// Mitsubishi GX Works2 project: pr6   PLC: Q03UDV

PROGRAM MAIN
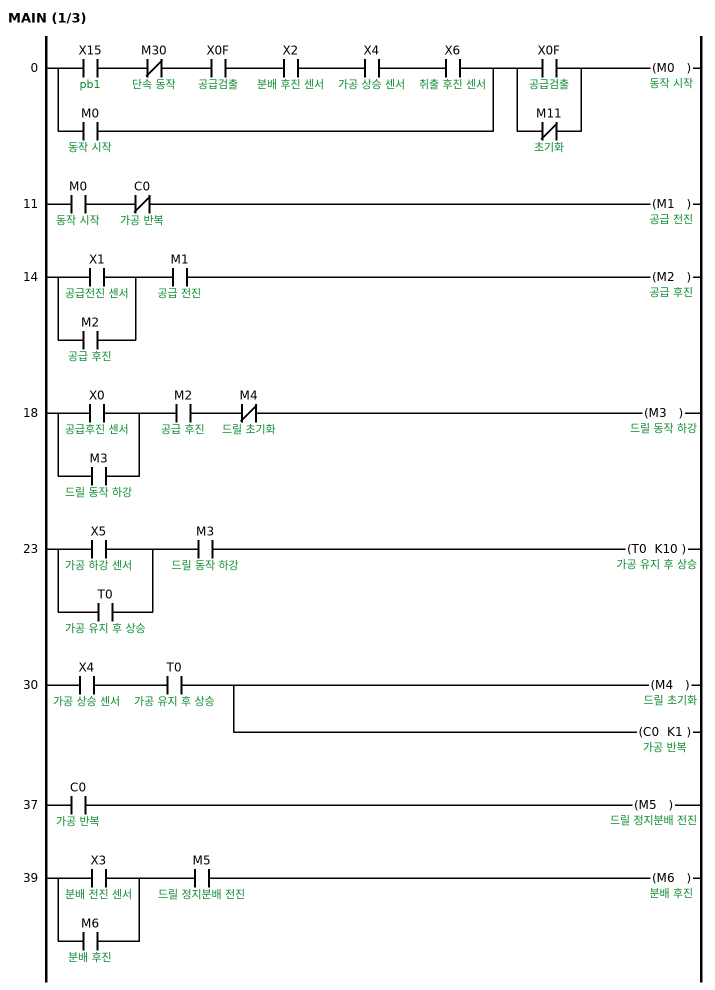
0     LD      X15  ; pb1
      ANI     M30  ; 단속 동작
      AND     X0F  ; 공급검출
      AND     X2  ; 분배 후진 센서
      AND     X4  ; 가공 상승 센서
      AND     X6  ; 취출 후진 센서
      OR      M0  ; 동작 시작
      LD      X0F  ; 공급검출
      ORI     M11  ; 초기화
      ANB
      OUT     M0  ; 동작 시작
11    LD      M0  ; 동작 시작
      ANI     C0  ; 가공 반복
      OUT     M1  ; 공급 전진
14    LD      X1  ; 공급전진 센서
      OR      M2  ; 공급 후진
      AND     M1  ; 공급 전진
      OUT     M2  ; 공급 후진
18    LD      X0  ; 공급후진 센서
      OR      M3  ; 드릴 동작 하강
      AND     M2  ; 공급 후진
      ANI     M4  ; 드릴 초기화
      OUT     M3  ; 드릴 동작 하강
23    LD      X5  ; 가공 하강 센서
      OR      T0  ; 가공 유지 후 상승
      AND     M3  ; 드릴 동작 하강
      OUT     T0 K10  ; 가공 유지 후 상승
30    LD      X4  ; 가공 상승 센서
      AND     T0  ; 가공 유지 후 상승
      OUT     M4  ; 드릴 초기화
      OUT     C0 K1  ; 가공 반복
37    LD      C0  ; 가공 반복
      OUT     M5  ; 드릴 정지분배 전진
39    LD      X3  ; 분배 전진 센서
      OR      M6  ; 분배 후진
      AND     M5  ; 드릴 정지분배 전진
      OUT     M6  ; 분배 후진
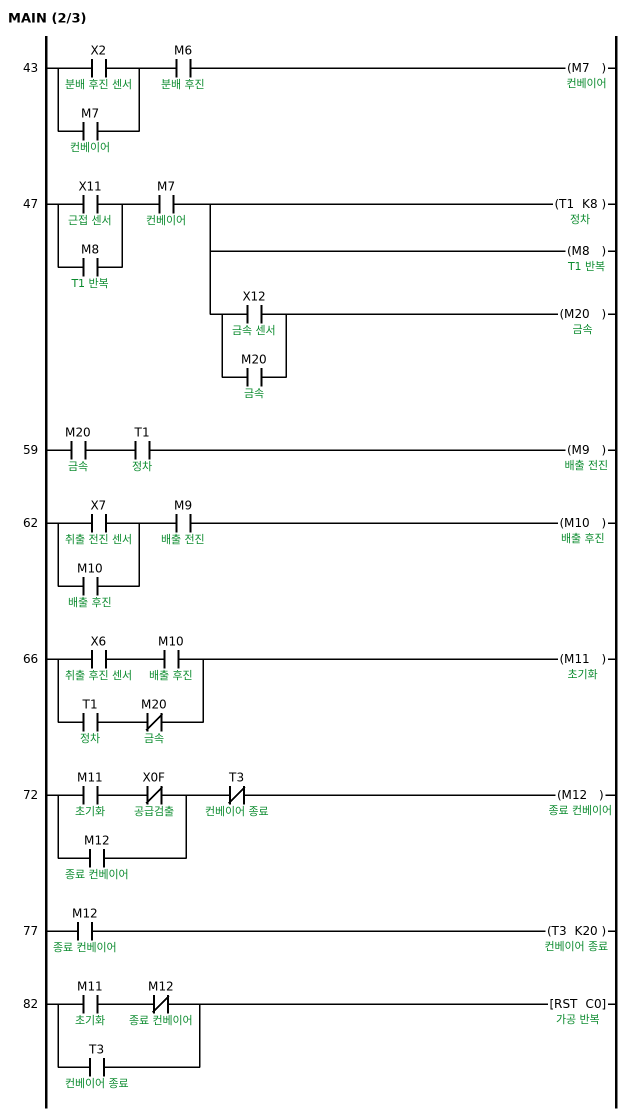
43    LD      X2  ; 분배 후진 센서
      OR      M7  ; 컨베이어
      AND     M6  ; 분배 후진
      OUT     M7  ; 컨베이어
47    LD      X11  ; 근접 센서
      OR      M8  ; T1 반복
      AND     M7  ; 컨베이어
      OUT     T1 K8  ; 정차
      OUT     M8  ; T1 반복
      LD      X12  ; 금속 센서
      OR      M20  ; 금속
      ANB
      OUT     M20  ; 금속
59    LD      M20  ; 금속
      AND     T1  ; 정차
      OUT     M9  ; 배출 전진
62    LD      X7  ; 취출 전진 센서
      OR      M10  ; 배출 후진
      AND     M9  ; 배출 전진
      OUT     M10  ; 배출 후진
66    LD      X6  ; 취출 후진 센서
      AND     M10  ; 배출 후진
      LD      T1  ; 정차
      ANI     M20  ; 금속
      ORB
      OUT     M11  ; 초기화
72    LD      M11  ; 초기화
      ANI     X0F  ; 공급검출
      OR      M12  ; 종료 컨베이어
      ANI     T3  ; 컨베이어 종료
      OUT     M12  ; 종료 컨베이어
77    LD      M12  ; 종료 컨베이어
      OUT     T3 K20  ; 컨베이어 종료
82    LD      M11  ; 초기화
      ANI     M12  ; 종료 컨베이어
      OR      T3  ; 컨베이어 종료
      RST     C0  ; 가공 반복
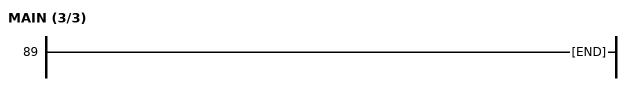
89    END
END_PROGRAM

PROGRAM OUTPUT
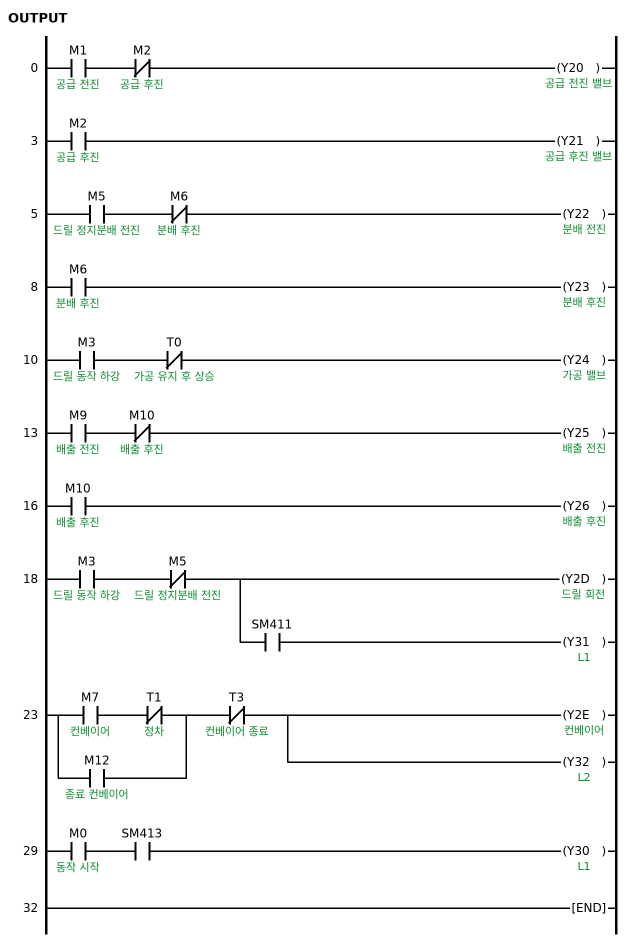
0     LD      M1  ; 공급 전진
      ANI     M2  ; 공급 후진
      OUT     Y20  ; 공급 전진 밸브
3     LD      M2  ; 공급 후진
      OUT     Y21  ; 공급 후진 밸브
5     LD      M5  ; 드릴 정지분배 전진
      ANI     M6  ; 분배 후진
      OUT     Y22  ; 분배 전진
8     LD      M6  ; 분배 후진
      OUT     Y23  ; 분배 후진
10    LD      M3  ; 드릴 동작 하강
      ANI     T0  ; 가공 유지 후 상승
      OUT     Y24  ; 가공 밸브
13    LD      M9  ; 배출 전진
      ANI     M10  ; 배출 후진
      OUT     Y25  ; 배출 전진
16    LD      M10  ; 배출 후진
      OUT     Y26  ; 배출 후진
18    LD      M3  ; 드릴 동작 하강
      ANI     M5  ; 드릴 정지분배 전진
      OUT     Y2D  ; 드릴 회전
      AND     SM411
      OUT     Y31  ; L1
23    LD      M7  ; 컨베이어
      ANI     T1  ; 정차
      OR      M12  ; 종료 컨베이어
      ANI     T3  ; 컨베이어 종료
      OUT     Y2E  ; 컨베이어
      OUT     Y32  ; L2
29    LD      M0  ; 동작 시작
      AND     SM413
      OUT     Y30  ; L1
32    END
END_PROGRAM

// device comments not shown above
X10  ; 근접 센서
X16  ; PB2
X18  ; pb4
M15  ; 초기화 묶음
M21  ; 프로그램 초기화
M40  ; 종료 버튼
M41  ; 종료조건
M100  ; 종료 버튼 눌림
M101  ; 전체 종료
T2  ; 드릴 유지
T4  ; 취출 복귀
T5  ; 컨베이어 정지
T10  ; 배출 전진
T20  ; 컨베이어 종료
C1  ; 반복 1
